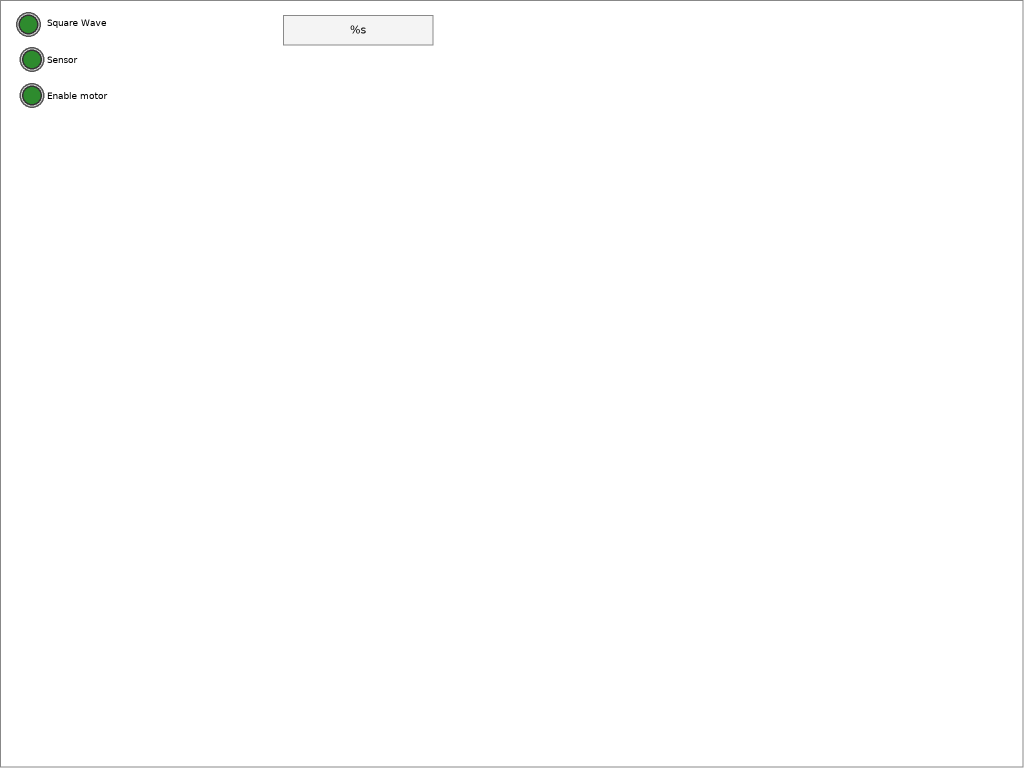
VISUALIZATION V_Main  // 1024x768
    Lamp1 (13,10 31x29), variable: DataExchange.bVar1, style: Lamp-Lamp1-Green
    Lamp1 (13,45 38x29), variable: DataExchange.sensor1, style: Lamp-Lamp1-Green
    Label (44,8 150x30), "Square Wave"
    Label (44,45 150x30), "Sensor"
    Lamp1 (13,81 38x29), variable: DataExchange.motor1, style: Lamp-Lamp1-Green
    Label (44,81 150x30), "Enable motor"
    Scrollbar (283,15 150x30), "%s", text variable: DataExchange.iVar1
        p1057716461: DataExchange.iVar1
END_VISUALIZATION

(* stored: Version 1.1.0.1, ProductVersion 3.1.4022.18
   Visu V_Main: Id {fb5ef48c-5d8c-4951-8413-81e7e18bd488} *)
